TYPE E_SendStates :
(**************************************************************************************
 * 	AUTHOR		Swisslog
 * 	LIBRARY		Data types/02_Library/02_Communication/TCP-Driver
 *	RELEASE		1.0.0
 * ------------------------------------------------------------------------------------
 * 	Revision History: 
 *
 * 	VERSION		DATE		INITIALS	DESCRIPTION
 *	0.1		07.09.2011	swl		initial version
 **************************************************************************************)
(
	SEND_IDLE,
	SEND_WAIT,
	SEND_ERROR
);
END_TYPE

(* stored: Version 1.1.0.1, ProductVersion 3.1.4020.6
   DUT E_SendStates: Id {717d4d2a-267a-4018-afb1-ca143fd2780c} *)
